(* IEC 61131-3 sources: OT-Security-Lab/plc, 3 files *)

(* ---- distribution.st ---- *)
// Distribution Process Logic (OpenPLC v4 ST project)
// Manages the distribution pump and discharge pressure.
//
// Build:  plc/build.sh   (compiled by STruC++ into plc/programs/distribution/program.zip)
// Register map (Modbus Holding Registers):
//   %QW0: Distribution pump command (0 = off, 1 = on)
//   %QW1: Discharge pressure (bar) - process state
//   %QW2: Pump speed (%)
//   %QW5: Pump runtime (hours) - accumulated
//   %QW6: Pressure alarm (0 = normal, 1 = low pressure with pump on)

PROGRAM MAIN
VAR
    PumpCommand   AT %QW0 : UINT;
    DischargePres AT %QW1 : UINT;
    PumpSpeed     AT %QW2 : UINT;
    PumpRuntime   AT %QW5 : UINT;
    PressureAlarm AT %QW6 : UINT;
END_VAR

// Process simulation: pressure follows pump state
IF PumpCommand = 1 THEN
    DischargePres := DischargePres + 1;
    PumpRuntime := PumpRuntime + 1;
    PumpSpeed := 80;
ELSE
    IF DischargePres >= 2 THEN
        DischargePres := DischargePres - 2;
    ELSE
        DischargePres := 0;
    END_IF;
    PumpSpeed := 0;
END_IF;

IF DischargePres > 10 THEN
    DischargePres := 10;
END_IF;

// Alarm: pump running but no pressure = failed pump / sabotage indicator
IF PumpCommand = 1 AND DischargePres < 2 THEN
    PressureAlarm := 1;
ELSE
    PressureAlarm := 0;
END_IF;

END_PROGRAM

CONFIGURATION Config0
  RESOURCE Res0 ON PLC
    TASK Task0(INTERVAL := T#500ms, PRIORITY := 0);
    PROGRAM Inst0 WITH Task0 : MAIN;
  END_RESOURCE
END_CONFIGURATION

(* ---- intake.st ---- *)
// Intake Process Logic (OpenPLC v4 ST project)
// Simulates the water intake tank and enforces the overflow safety interlock.
//
// Build:  plc/build.sh   (compiled by STruC++ into plc/programs/intake/program.zip)
// Register map (Modbus Holding Registers):
//   %QW0: Inlet Valve command (0 = closed, 1 = open)
//   %QW1: Intake pump speed (%)
//   %QW5: Tank Level (%) - process state, simulated here
//   %QW6: Interlock alarm (0 = normal, 1 = overflow interlock tripped)

PROGRAM MAIN
VAR
    InletValve AT %QW0 : UINT;
    Pump       AT %QW1 : UINT;
    TankLevel  AT %QW5 : UINT;
    Alarm      AT %QW6 : UINT;
END_VAR

// --- Process simulation: autonomous level control ---
// A real intake station keeps the tank within an operating band. The level
// controller calls for water when the tank is low; the SIS interlock (below)
// is the independent high-high trip at 95%.
IF TankLevel < 20 THEN
    InletValve := 1;
END_IF;

IF InletValve = 1 THEN
    // Filling: level rises while the inlet valve is open
    TankLevel := TankLevel + 1;
ELSE
    // Draining: level falls when the valve is closed
    TankLevel := TankLevel - 1;
END_IF;

IF TankLevel > 100 THEN
    TankLevel := 100;
END_IF;

IF TankLevel < 0 THEN
    TankLevel := 0;
END_IF;

// --- Safety interlock (IEC 61511 SIS-style) ---
// Hard override: never allow the inlet valve to remain open above 95% level.
// The network-side IDS shadows a tighter 90% envelope for defense in depth.
IF TankLevel > 95 THEN
    InletValve := 0;
    Alarm := 1;
ELSE
    Alarm := 0;
END_IF;

END_PROGRAM

CONFIGURATION Config0
  RESOURCE Res0 ON PLC
    TASK Task0(INTERVAL := T#500ms, PRIORITY := 0);
    PROGRAM Inst0 WITH Task0 : MAIN;
  END_RESOURCE
END_CONFIGURATION

(* ---- treatment.st ---- *)
// Treatment Process Logic (OpenPLC v4 ST project)
// Controls chemical dosing based on incoming flow.
//
// Build:  plc/build.sh   (compiled by STruC++ into plc/programs/treatment/program.zip)
// Register map (Modbus Holding Registers):
//   %QW0: Inlet flow (m3/h) - process state
//   %QW1: Dosing pump command (0 = off, 1 = on)
//   %QW2: Dosing rate (%)
//   %QW5: Residual chlorine (ppm) - process state
//   %QW6: Dosing alarm (0 = normal, 1 = out-of-range)

PROGRAM MAIN
VAR
    InletFlow      AT %QW0 : UINT;
    DosingPump     AT %QW1 : UINT;
    DosingRate     AT %QW2 : UINT;
    ResidualChlor  AT %QW5 : UINT;
    DosingAlarm    AT %QW6 : UINT;
END_VAR

// Process simulation: residual chlorine decays over time
IF ResidualChlor > 0 THEN
    ResidualChlor := ResidualChlor - 1;
END_IF;

// Dosing control: pump engages when flow is present and chlorine is low
IF InletFlow > 0 AND ResidualChlor < 20 THEN
    DosingPump := 1;
    DosingRate := 50;
ELSIF ResidualChlor >= 40 THEN
    DosingPump := 0;
    DosingRate := 0;
END_IF;

// Out-of-range chlorine is a process alarm
IF ResidualChlor > 60 OR (InletFlow > 0 AND ResidualChlor = 0) THEN
    DosingAlarm := 1;
ELSE
    DosingAlarm := 0;
END_IF;

END_PROGRAM

CONFIGURATION Config0
  RESOURCE Res0 ON PLC
    TASK Task0(INTERVAL := T#500ms, PRIORITY := 0);
    PROGRAM Inst0 WITH Task0 : MAIN;
  END_RESOURCE
END_CONFIGURATION
